Fanuc KAREL source: ks00024.KL

PROGRAM KS00024
%STACKSIZE=65535
%PRIORITY=65535
%NOLOCKGROUP
VAR
FLAG : BOOLEAN
N : INTEGER
STATUS : INTEGER
PN : STRING[80]
VN : STRING[80]
-- UNRESOLVED DECLARATIONS (source type spelling not recovered)
-- A : TYPE_0x1101 (type_u16=0x1101)
-- B : TYPE_0x1101 (type_u16=0x1101)
BEGIN
PN=''
VN='A'
-- UNRESOLVED_PC line 19 opcodes [22 22 30] marker_code=27
END KS00024
